{attribute 'linkalways'} 
{attribute 'no_explicit_call' := 'This FB is a CLASS and must be accessed using methods or properties'}
{attribute 'enable_dynamic_creation'}
FUNCTION_BLOCK _TcVnVector4_DINT EXTENDS AliasDatatypeBase
VAR
	localData : TcVnVector4_DINT;
	activeData : REFERENCE TO TcVnVector4_DINT REF= localData;
	aliasBaseDatatype : _Array0to3OfDINT;
END_VAR

PROPERTY PUBLIC Address : PVOID
GET
Address := ADR(activeData);
END_GET
END_PROPERTY

METHOD PUBLIC ClearReference
VAR_INPUT
END_VAR
activeData REF= localData;
SetBaseDatatypeReference();
END_METHOD

METHOD PUBLIC Clone : I_Datatype
VAR
    pClone : POINTER TO _TcVnVector4_DINT;
END_VAR
pClone := __NEW(_TcVnVector4_DINT);
Clone := pClone^;
END_METHOD

METHOD FB_init : BOOL
VAR_INPUT
	bInitRetains : BOOL; // if TRUE, the retain variables are initialized (warm start / cold start)
	bInCopyCode : BOOL;  // if TRUE, the instance afterwards gets moved into the copy code (online change)
	//InitialValue : <type>; // if possible, not all values can be initialized
END_VAR
//localData := InitialValue; // if possible, not all values can be initialized
SetBaseDatatypeReference();
AddBaseDatatype(aliasBaseDatatype);
END_METHOD

PROPERTY PUBLIC Identifier : T_MAXSTRING
GET
Identifier := 'TcVnVector4_DINT';
END_GET
END_PROPERTY

METHOD PUBLIC MakeReferenceTo
VAR_INPUT
	ReferenceTarget : REFERENCE TO TcVnVector4_DINT;
END_VAR
activeData REF= ReferenceTarget;
SetBaseDatatypeReference();
END_METHOD

METHOD PROTECTED SetBaseDatatypeReference
VAR_INPUT
END_VAR
aliasBaseDatatype.MakeReferenceTo(activeData);
END_METHOD

PROPERTY PUBLIC Size : UDINT
GET
Size := SIZEOF(activeData);
END_GET
END_PROPERTY

METHOD TryMakeReferenceTo : BOOL
VAR_INPUT
	Target : I_Datatype;
END_VAR
VAR
	targetAsAlias : I_AliasDatatype;
	pTargetData : POINTER TO TcVnVector4_DINT;
END_VAR
IF NOT Target.TryResolveAsAliasDatatype(targetAsAlias) THEN
	RETURN;
END_IF

IF targetAsAlias.Identifier <> Identifier THEN
	RETURN;
END_IF

pTargetData := Target.Address;
activeData REF= pTargetData^;
SetBaseDatatypeReference();
TryMakeReferenceTo := TRUE;
END_METHOD

PROPERTY PUBLIC Value : REFERENCE TO TcVnVector4_DINT
GET
Value REF= activeData;
END_GET
END_PROPERTY

END_FUNCTION_BLOCK

(* stored: Version 1.1.0.1, ProductVersion 3.1.4024.13
   POU _TcVnVector4_DINT: Id {d752e18c-2e38-08be-1160-0f3a0d764aa9}, SpecialFunc None
   Folder Core: Id {596beb3b-0e2d-0c78-104c-51f37453fd66}
   Folder Protected: Id {19c4753f-3ed4-04b1-3d1b-bc1284bd7bea}
   Folder Customize: Id {e33041c7-0dfd-0086-1772-271561566b25}
   Folder Constructor: Id {ce00d6f8-0359-06ec-0087-0567963a902b}
   Property Address: Id {e63b299d-62a5-0d89-189d-b49c456ab848}
   Get Get: Id {d97c45d4-f673-05c1-3d3b-cedba50cf161}
   Method ClearReference: Id {abb9a07a-efd2-0da0-2a68-20f1c246a07d}
   Method Clone: Id {96d551fe-e949-0b30-19fe-b65d2b9e741f}
   Method FB_init: Id {138c3f41-45d3-0508-1ae8-621d5529d97c}
   Property Identifier: Id {81067726-e7e8-0e9c-14c2-7db014b5fc2d}
   Get Get: Id {1616835a-7e60-07f4-0c5d-9a52f0d292c5}
   Method MakeReferenceTo: Id {bd9f73d8-a575-0f79-34cb-a2ab4d1a6d30}
   Method SetBaseDatatypeReference: Id {3a228502-cdf0-0832-0aa3-4c4017de0aca}
   Property Size: Id {779ee175-229e-0691-3d76-56eaced093fd}
   Get Get: Id {32e9bf83-5365-0db7-1bff-1e70e61135c2}
   Method TryMakeReferenceTo: Id {b9466735-42df-0f4c-3e64-0543364cc1b6}
   Property Value: Id {a36ace49-81cc-0fbb-06c9-116af9c68c2c}
   Get Get: Id {522405e8-d651-0816-14cf-4d9f070ca493} *)
